PROGRAM MAIN
VAR
END_VAR

;

END_PROGRAM

(* stored: Version 1.0
   POU MAIN: Id {00000000-0000-0000-0000-000000000000} *)
